LIN {X 0,Y 84.435,Z 449.066,A -85,B 0,C 180,E1 -28060.558,E2 -28060.558} C_VEL
LIN {X 0,Y 93.266,Z 446.921,A -85,B 0,C 180,E1 -28068.394,E2 -28068.394} C_VEL
LIN {X 0,Y 102.413,Z 443.94,A -85,B 0,C 180,E1 -28074.267,E2 -28074.267} C_VEL
LIN {X 0,Y 114.487,Z 439.001,A -85,B 0,C 180,E1 -28080.004,E2 -28080.004} C_VEL
LIN {X 0,Y 126.871,Z 432.782,A -85,B 0,C 180,E1 -28084.39,E2 -28084.39} C_VEL
LIN {X 0,Y 138.251,Z 425.939,A -85,B 0,C 180,E1 -28087.588,E2 -28087.588} C_VEL
LIN {X 0,Y 142.198,Z 423.34,A -85,B 0,C 180,E1 -28088.53,E2 -28088.53} C_VEL
LIN {X 0,Y 144.172,Z 421.915,A -85,B 0,C 180,E1 -28089.196,E2 -28089.196} C_VEL
LIN {X 0,Y 144.424,Z 421.642,A -85,B 0,C 180,E1 -28091.227,E2 -28091.227} C_VEL
LIN {X 0,Y 144.055,Z 421.993,A -85,B 0,C 180,E1 -28094.122,E2 -28094.122} C_VEL
LIN {X 0,Y 143.259,Z 423.001,A -85,B 0,C 180,E1 -28097.121,E2 -28097.121} C_VEL
LIN {X 0,Y 142.165,Z 424.543,A -85,B 0,C 180,E1 -28100.249,E2 -28100.249} C_VEL
LIN {X 0,Y 139.969,Z 426.46,A -85,B 0,C 180,E1 -28101.741,E2 -28101.741} C_VEL
LIN {X 0,Y 127.709,Z 434.572,A -85,B 0,C 180,E1 -28104.773,E2 -28104.773} C_VEL
LIN {X 0,Y 115.927,Z 441.264,A -85,B 0,C 180,E1 -28108.477,E2 -28108.477} C_VEL
LIN {X 0,Y 104.888,Z 446.652,A -85,B 0,C 180,E1 -28113.122,E2 -28113.122} C_VEL
LIN {X 0,Y 97.213,Z 449.956,A -85,B 0,C 180,E1 -28117.326,E2 -28117.326} C_VEL
LIN {X 0,Y 87.921,Z 453.371,A -85,B 0,C 180,E1 -28123.998,E2 -28123.998} C_VEL
LIN {X 0,Y 80.134,Z 455.727,A -85,B 0,C 180,E1 -28132.131,E2 -28132.131} C_VEL
LIN {X 0,Y 74.339,Z 457.09,A -85,B 0,C 180,E1 -28141.795,E2 -28141.795} C_VEL
LIN {X 0,Y 70.967,Z 457.423,A -85,B 0,C 180,E1 -28152.721,E2 -28152.721} C_VEL
LIN {X 0,Y 70.115,Z 456.671,A -85,B 0,C 180,E1 -28164.251,E2 -28164.251} C_VEL
LIN {X 0,Y 70.375,Z 455.877,A -85,B 0,C 180,E1 -28170.004,E2 -28170.004} C_VEL
LIN {X 0,Y 70.197,Z 454.698,A -85,B 0,C 180,E1 -28175.75,E2 -28175.75} C_VEL
LIN {X 0,Y 71.141,Z 451.341,A -85,B 0,C 180,E1 -28187.244,E2 -28187.244} C_VEL
LIN {X 0,Y 74.509,Z 446.636,A -85,B 0,C 180,E1 -28198.143,E2 -28198.143} C_VEL
LIN {X 0,Y 80.106,Z 440.454,A -85,B 0,C 180,E1 -28207.893,E2 -28207.893} C_VEL
LIN {X 0,Y 87.693,Z 432.656,A -85,B 0,C 180,E1 -28216.165,E2 -28216.165} C_VEL
LIN {X 0,Y 95.422,Z 424.288,A -85,B 0,C 180,E1 -28222.354,E2 -28222.354} C_VEL
LIN {X 0,Y 104.607,Z 413.774,A -85,B 0,C 180,E1 -28227.655,E2 -28227.655} C_VEL
LIN {X 0,Y 109.555,Z 407.579,A -85,B 0,C 180,E1 -28230.005,E2 -28230.005} C_VEL
LIN {X 0,Y 111.039,Z 404.584,A -85,B 0,C 180,E1 -28231.43,E2 -28231.43} C_VEL
LIN {X 0,Y 114.396,Z 395.038,A -85,B 0,C 180,E1 -28236.106,E2 -28236.106} C_VEL
LIN {X 0,Y 115,Z 392.347,A -85,B 0,C 180,E1 -28237.541,E2 -28237.541} C_VEL
LIN {X 0,Y 115.079,Z 383.981,A -85,B 0,C 180,E1 -28243.133,E2 -28243.133} C_VEL
LIN {X 0,Y 114.938,Z 378.464,A -85,B 0,C 180,E1 -28247.035,E2 -28247.035} C_VEL
LIN {X 0,Y 114.63,Z 373.213,A -85,B 0,C 180,E1 -28251.18,E2 -28251.18} C_VEL
LIN {X 0,Y 114.056,Z 367.486,A -85,B 0,C 180,E1 -28256.464,E2 -28256.464} C_VEL
LIN {X 0,Y 113.576,Z 364.537,A -85,B 0,C 180,E1 -28259.996,E2 -28259.996} C_VEL
LIN {X 0,Y 112.79,Z 361.934,A -85,B 0,C 180,E1 -28264.434,E2 -28264.434} C_VEL
LIN {X 0,Y 111.583,Z 360.171,A -85,B 0,C 180,E1 -28270.888,E2 -28270.888} C_VEL
LIN {X 0,Y 111.233,Z 359.571,A -85,B 0,C 180,E1 -28274.635,E2 -28274.635} C_VEL
LIN {X 0,Y 110.968,Z 359.662,A -85,B 0,C 180,E1 -28278.457,E2 -28278.457} C_VEL
LIN {X 0,Y 111.036,Z 361.087,A -85,B 0,C 180,E1 -28286.295,E2 -28286.295} C_VEL
LIN {X 0,Y 111.487,Z 362.203,A -85,B 0,C 180,E1 -28290.281,E2 -28290.281} C_VEL
LIN {X 0,Y 112.237,Z 364.789,A -85,B 0,C 180,E1 -28295.505,E2 -28295.505} C_VEL
LIN {X 0,Y 113.399,Z 369.059,A -85,B 0,C 180,E1 -28301.948,E2 -28301.948} C_VEL
LIN {X 0,Y 114.267,Z 372.788,A -85,B 0,C 180,E1 -28306.337,E2 -28306.337} C_VEL
LIN {X 0,Y 115.456,Z 378.791,A -85,B 0,C 180,E1 -28312.303,E2 -28312.303} C_VEL
LIN {X 0,Y 116.307,Z 385.128,A -85,B 0,C 180,E1 -28317.768,E2 -28317.768} C_VEL
LIN {X 0,Y 116.576,Z 388.345,A -85,B 0,C 180,E1 -28320.283,E2 -28320.283} C_VEL
LIN {X 0,Y 115.982,Z 390.167,A -85,B 0,C 180,E1 -28321.236,E2 -28321.236} C_VEL
LIN {X 0,Y 114.077,Z 392.752,A -85,B 0,C 180,E1 -28321.917,E2 -28321.917} C_VEL
LIN {X 0,Y 111.26,Z 395.53,A -85,B 0,C 180,E1 -28322.257,E2 -28322.257} C_VEL
LIN {X 0,Y 105.593,Z 400.429,A -85,B 0,C 180,E1 -28322.611,E2 -28322.611} C_VEL
LIN {X 0,Y 102.68,Z 403.357,A -85,B 0,C 180,E1 -28323.39,E2 -28323.39} C_VEL
LIN {X 0,Y 93.99,Z 413.25,A -85,B 0,C 180,E1 -28328.043,E2 -28328.043} C_VEL
LIN {X 0,Y 84.929,Z 422.622,A -85,B 0,C 180,E1 -28334.395,E2 -28334.395} C_VEL
LIN {X 0,Y 76.825,Z 430.56,A -85,B 0,C 180,E1 -28342.404,E2 -28342.404} C_VEL
LIN {X 0,Y 70.311,Z 436.93,A -85,B 0,C 180,E1 -28351.925,E2 -28351.925} C_VEL
LIN {X 0,Y 65.767,Z 441.73,A -85,B 0,C 180,E1 -28362.336,E2 -28362.336} C_VEL
LIN {X 0,Y 63.881,Z 444.105,A -85,B 0,C 180,E1 -28369.267,E2 -28369.267} C_VEL
LIN {X 0,Y 62.766,Z 446.112,A -85,B 0,C 180,E1 -28376.603,E2 -28376.603} C_VEL
LIN {X 0,Y 62.801,Z 448.526,A -85,B 0,C 180,E1 -28388.442,E2 -28388.442} C_VEL
LIN {X 0,Y 64.853,Z 449.915,A -85,B 0,C 180,E1 -28399.452,E2 -28399.452} C_VEL
LIN {X 0,Y 68.561,Z 450.524,A -85,B 0,C 180,E1 -28409.175,E2 -28409.175} C_VEL
LIN {X 0,Y 75.079,Z 450.236,A -85,B 0,C 180,E1 -28419.392,E2 -28419.392} C_VEL
LIN {X 0,Y 80.094,Z 449.536,A -85,B 0,C 180,E1 -28424.83,E2 -28424.83} C_VEL
LIN {X 0,Y 87.142,Z 448.045,A -85,B 0,C 180,E1 -28430.723,E2 -28430.723} C_VEL
LIN {X 0,Y 98.471,Z 444.801,A -85,B 0,C 180,E1 -28437.627,E2 -28437.627} C_VEL
LIN {X 0,Y 108.834,Z 441.008,A -85,B 0,C 180,E1 -28442.271,E2 -28442.271} C_VEL
LIN {X 0,Y 121.685,Z 435.179,A -85,B 0,C 180,E1 -28446.637,E2 -28446.637} C_VEL
LIN {X 0,Y 133.12,Z 428.918,A -85,B 0,C 180,E1 -28449.679,E2 -28449.679} C_VEL
LIN {X 0,Y 138.452,Z 425.626,A -85,B 0,C 180,E1 -28450.902,E2 -28450.902} C_VEL
LIN {X 0,Y 138.46,Z 425.624,A -85,B 0,C 180,E1 -28451.717,E2 -28451.717} C_VEL
LIN {X 0,Y 137.869,Z 426.196,A -85,B 0,C 180,E1 -28454.769,E2 -28454.769} C_VEL
LIN {X 0,Y 136.829,Z 427.379,A -85,B 0,C 180,E1 -28457.953,E2 -28457.953} C_VEL
LIN {X 0,Y 136.23,Z 428.01,A -85,B 0,C 180,E1 -28459.101,E2 -28459.101} C_VEL
LIN {X 0,Y 134.35,Z 429.323,A -85,B 0,C 180,E1 -28459.685,E2 -28459.685} C_VEL
LIN {X 0,Y 121.815,Z 436.836,A -85,B 0,C 180,E1 -28462.622,E2 -28462.622} C_VEL
LIN {X 0,Y 109.748,Z 442.965,A -85,B 0,C 180,E1 -28466.301,E2 -28466.301} C_VEL
LIN {X 0,Y 98.408,Z 447.887,A -85,B 0,C 180,E1 -28471.024,E2 -28471.024} C_VEL
LIN {X 0,Y 87.892,Z 451.729,A -85,B 0,C 180,E1 -28476.912,E2 -28476.912} C_VEL
LIN {X 0,Y 78.624,Z 454.487,A -85,B 0,C 180,E1 -28484.354,E2 -28484.354} C_VEL
LIN {X 0,Y 71.075,Z 456.19,A -85,B 0,C 180,E1 -28493.614,E2 -28493.614} C_VEL
LIN {X 0,Y 65.75,Z 456.915,A -85,B 0,C 180,E1 -28504.692,E2 -28504.692} C_VEL
LIN {X 0,Y 63.244,Z 456.628,A -85,B 0,C 180,E1 -28517.163,E2 -28517.163} C_VEL
LIN {X 0,Y 63.269,Z 455.362,A -85,B 0,C 180,E1 -28528.967,E2 -28528.967} C_VEL
LIN {X 0,Y 63.278,Z 454.973,A -85,B 0,C 180,E1 -28531.435,E2 -28531.435} C_VEL
LIN {X 0,Y 63.36,Z 452.358,A -85,B 0,C 180,E1 -28542.822,E2 -28542.822} C_VEL
LIN {X 0,Y 65.962,Z 448.192,A -85,B 0,C 180,E1 -28555.23,E2 -28555.23} C_VEL
LIN {X 0,Y 71.113,Z 442.605,A -85,B 0,C 180,E1 -28566.373,E2 -28566.373} C_VEL
LIN {X 0,Y 78.493,Z 435.471,A -85,B 0,C 180,E1 -28575.754,E2 -28575.754} C_VEL
LIN {X 0,Y 86.318,Z 427.807,A -85,B 0,C 180,E1 -28582.551,E2 -28582.551} C_VEL
LIN {X 0,Y 95.096,Z 418.555,A -85,B 0,C 180,E1 -28588.206,E2 -28588.206} C_VEL
LIN {X 0,Y 103.318,Z 409.184,A -85,B 0,C 180,E1 -28592.171,E2 -28592.171} C_VEL
LIN {X 0,Y 104.666,Z 407.393,A -85,B 0,C 180,E1 -28592.84,E2 -28592.84} C_VEL
LIN {X 0,Y 108.113,Z 399.375,A -85,B 0,C 180,E1 -28597.039,E2 -28597.039} C_VEL
LIN {X 0,Y 109.02,Z 397.059,A -85,B 0,C 180,E1 -28598.239,E2 -28598.239} C_VEL
LIN {X 0,Y 109.45,Z 395.202,A -85,B 0,C 180,E1 -28599.315,E2 -28599.315} C_VEL
LIN {X 0,Y 109.816,Z 389.011,A -85,B 0,C 180,E1 -28603.743,E2 -28603.743} C_VEL
LIN {X 0,Y 110.07,Z 382.163,A -85,B 0,C 180,E1 -28608.953,E2 -28608.953} C_VEL
LIN {X 0,Y 110.062,Z 377.813,A -85,B 0,C 180,E1 -28612.659,E2 -28612.659} C_VEL
LIN {X 0,Y 109.848,Z 372.283,A -85,B 0,C 180,E1 -28618.163,E2 -28618.163} C_VEL
LIN {X 0,Y 109.497,Z 369.596,A -85,B 0,C 180,E1 -28621.835,E2 -28621.835} C_VEL
LIN {X 0,Y 109.263,Z 368.507,A -85,B 0,C 180,E1 -28623.684,E2 -28623.684} C_VEL
LIN {X 0,Y 108.568,Z 367.207,A -85,B 0,C 180,E1 -28627.435,E2 -28627.435} C_VEL
LIN {X 0,Y 107.907,Z 366.105,A -85,B 0,C 180,E1 -28632.314,E2 -28632.314} C_VEL
LIN {X 0,Y 107.692,Z 365.766,A -85,B 0,C 180,E1 -28635.127,E2 -28635.127} C_VEL
LIN {X 0,Y 107.409,Z 365.93,A -85,B 0,C 180,E1 -28639.092,E2 -28639.092} C_VEL
LIN {X 0,Y 107.5,Z 367.459,A -85,B 0,C 180,E1 -28647.23,E2 -28647.23} C_VEL
LIN {X 0,Y 107.884,Z 369.197,A -85,B 0,C 180,E1 -28652.122,E2 -28652.122} C_VEL
LIN {X 0,Y 108.479,Z 371.709,A -85,B 0,C 180,E1 -28656.933,E2 -28656.933} C_VEL
LIN {X 0,Y 109.142,Z 375.046,A -85,B 0,C 180,E1 -28661.98,E2 -28661.98} C_VEL
LIN {X 0,Y 109.866,Z 379.541,A -85,B 0,C 180,E1 -28667.352,E2 -28667.352} C_VEL
LIN {X 0,Y 110.51,Z 384.899,A -85,B 0,C 180,E1 -28672.788,E2 -28672.788} C_VEL
LIN {X 0,Y 110.898,Z 390.369,A -85,B 0,C 180,E1 -28677.745,E2 -28677.745} C_VEL
LIN {X 0,Y 110.948,Z 392.488,A -85,B 0,C 180,E1 -28679.549,E2 -28679.549} C_VEL
LIN {X 0,Y 106.792,Z 398.244,A -85,B 0,C 180,E1 -28681.499,E2 -28681.499} C_VEL
LIN {X 0,Y 102.68,Z 403.357,A -85,B 0,C 180,E1 -28683.39,E2 -28683.39} C_VEL
LIN {X 0,Y 98.976,Z 407.288,A -85,B 0,C 180,E1 -28684.753,E2 -28684.753} C_VEL
LIN {X 0,Y 91.631,Z 413.346,A -85,B 0,C 180,E1 -28686.431,E2 -28686.431} C_VEL
LIN {X 0,Y 84.102,Z 418.989,A -85,B 0,C 180,E1 -28688.532,E2 -28688.532} C_VEL
LIN {X 0,Y 80.223,Z 422.232,A -85,B 0,C 180,E1 -28690.666,E2 -28690.666} C_VEL
LIN {X 0,Y 71.548,Z 430.198,A -85,B 0,C 180,E1 -28698.666,E2 -28698.666} C_VEL
LIN {X 0,Y 65.295,Z 435.825,A -85,B 0,C 180,E1 -28706.911,E2 -28706.911} C_VEL
LIN {X 0,Y 60.404,Z 440.436,A -85,B 0,C 180,E1 -28716.677,E2 -28716.677} C_VEL
LIN {X 0,Y 56.94,Z 444.245,A -85,B 0,C 180,E1 -28727.968,E2 -28727.968} C_VEL
LIN {X 0,Y 55.419,Z 447.223,A -85,B 0,C 180,E1 -28740.476,E2 -28740.476} C_VEL
LIN {X 0,Y 55.969,Z 449.038,A -85,B 0,C 180,E1 -28751.126,E2 -28751.126} C_VEL
LIN {X 0,Y 59.505,Z 450.641,A -85,B 0,C 180,E1 -28765.758,E2 -28765.758} C_VEL
LIN {X 0,Y 63.082,Z 451.003,A -85,B 0,C 180,E1 -28773.544,E2 -28773.544} C_VEL
LIN {X 0,Y 68.931,Z 450.835,A -85,B 0,C 180,E1 -28782.196,E2 -28782.196} C_VEL
LIN {X 0,Y 78.225,Z 449.653,A -85,B 0,C 180,E1 -28791.195,E2 -28791.195} C_VEL
LIN {X 0,Y 84.571,Z 448.377,A -85,B 0,C 180,E1 -28795.683,E2 -28795.683} C_VEL
LIN {X 0,Y 92.271,Z 446.416,A -85,B 0,C 180,E1 -28800.005,E2 -28800.005} C_VEL
LIN {X 0,Y 101.268,Z 443.618,A -85,B 0,C 180,E1 -28803.984,E2 -28803.984} C_VEL
LIN {X 0,Y 113.609,Z 438.825,A -85,B 0,C 180,E1 -28808.217,E2 -28808.217} C_VEL
LIN {X 0,Y 127.424,Z 432.18,A -85,B 0,C 180,E1 -28811.777,E2 -28811.777} C_VEL
LIN {X 0,Y 130.443,Z 430.488,A -85,B 0,C 180,E1 -28812.449,E2 -28812.449} C_VEL
LIN {X 0,Y 132.034,Z 429.617,A -85,B 0,C 180,E1 -28813.258,E2 -28813.258} C_VEL
LIN {X 0,Y 131.347,Z 430.27,A -85,B 0,C 180,E1 -28815.616,E2 -28815.616} C_VEL
LIN {X 0,Y 130.943,Z 430.7,A -85,B 0,C 180,E1 -28816.9,E2 -28816.9} C_VEL
LIN {X 0,Y 122.449,Z 435.584,A -85,B 0,C 180,E1 -28818.741,E2 -28818.741} C_VEL
LIN {X 0,Y 109.858,Z 441.845,A -85,B 0,C 180,E1 -28821.941,E2 -28821.941} C_VEL
LIN {X 0,Y 97.812,Z 446.907,A -85,B 0,C 180,E1 -28826.091,E2 -28826.091} C_VEL
LIN {X 0,Y 83.782,Z 451.635,A -85,B 0,C 180,E1 -28832.988,E2 -28832.988} C_VEL
LIN {X 0,Y 73.799,Z 454.277,A -85,B 0,C 180,E1 -28840.378,E2 -28840.378} C_VEL
LIN {X 0,Y 65.432,Z 455.854,A -85,B 0,C 180,E1 -28849.881,E2 -28849.881} C_VEL
LIN {X 0,Y 59.347,Z 456.429,A -85,B 0,C 180,E1 -28861.732,E2 -28861.732} C_VEL
LIN {X 0,Y 56.308,Z 456.029,A -85,B 0,C 180,E1 -28875.55,E2 -28875.55} C_VEL
LIN {X 0,Y 55.963,Z 455.433,A -85,B 0,C 180,E1 -28882.791,E2 -28882.791} C_VEL
LIN {X 0,Y 56.231,Z 454.518,A -85,B 0,C 180,E1 -28890.005,E2 -28890.005} C_VEL
LIN {X 0,Y 56.012,Z 453.189,A -85,B 0,C 180,E1 -28897.213,E2 -28897.213} C_VEL
LIN {X 0,Y 57.652,Z 449.55,A -85,B 0,C 180,E1 -28911.456,E2 -28911.456} C_VEL
LIN {X 0,Y 62.206,Z 444.536,A -85,B 0,C 180,E1 -28924.4,E2 -28924.4} C_VEL
LIN {X 0,Y 69.338,Z 438.038,A -85,B 0,C 180,E1 -28935.2,E2 -28935.2} C_VEL
LIN {X 0,Y 78.408,Z 429.881,A -85,B 0,C 180,E1 -28943.781,E2 -28943.781} C_VEL
LIN {X 0,Y 87.349,Z 421.109,A -85,B 0,C 180,E1 -28949.881,E2 -28949.881} C_VEL
LIN {X 0,Y 97.253,Z 410.652,A -85,B 0,C 180,E1 -28954.598,E2 -28954.598} C_VEL
LIN {X 0,Y 98.701,Z 409.013,A -85,B 0,C 180,E1 -28955.215,E2 -28955.215} C_VEL
LIN {X 0,Y 99.978,Z 407.155,A -85,B 0,C 180,E1 -28956.048,E2 -28956.048} C_VEL
LIN {X 0,Y 103.355,Z 399.779,A -85,B 0,C 180,E1 -28960.119,E2 -28960.119} C_VEL
LIN {X 0,Y 103.926,Z 397.995,A -85,B 0,C 180,E1 -28961.226,E2 -28961.226} C_VEL
LIN {X 0,Y 104.85,Z 390.093,A -85,B 0,C 180,E1 -28967.414,E2 -28967.414} C_VEL
LIN {X 0,Y 105.332,Z 384.283,A -85,B 0,C 180,E1 -28972.327,E2 -28972.327} C_VEL
LIN {X 0,Y 105.52,Z 379.048,A -85,B 0,C 180,E1 -28977.56,E2 -28977.56} C_VEL
LIN {X 0,Y 105.567,Z 376.988,A -85,B 0,C 180,E1 -28979.996,E2 -28979.996} C_VEL
LIN {X 0,Y 105.304,Z 374.531,A -85,B 0,C 180,E1 -28983.823,E2 -28983.823} C_VEL
LIN {X 0,Y 104.738,Z 373.153,A -85,B 0,C 180,E1 -28987.708,E2 -28987.708} C_VEL
LIN {X 0,Y 104.24,Z 372.25,A -85,B 0,C 180,E1 -28991.665,E2 -28991.665} C_VEL
LIN {X 0,Y 103.9,Z 371.842,A -85,B 0,C 180,E1 -28995.694,E2 -28995.694} C_VEL
LIN {X 0,Y 103.586,Z 372.099,A -85,B 0,C 180,E1 -28999.826,E2 -28999.826} C_VEL
LIN {X 0,Y 103.496,Z 372.773,A -85,B 0,C 180,E1 -29004.039,E2 -29004.039} C_VEL
LIN {X 0,Y 103.646,Z 373.83,A -85,B 0,C 180,E1 -29008.332,E2 -29008.332} C_VEL
LIN {X 0,Y 103.869,Z 375.502,A -85,B 0,C 180,E1 -29012.767,E2 -29012.767} C_VEL
LIN {X 0,Y 104.28,Z 377.851,A -85,B 0,C 180,E1 -29017.335,E2 -29017.335} C_VEL
LIN {X 0,Y 104.682,Z 381.147,A -85,B 0,C 180,E1 -29022.392,E2 -29022.392} C_VEL
LIN {X 0,Y 105.064,Z 385.768,A -85,B 0,C 180,E1 -29028.012,E2 -29028.012} C_VEL
LIN {X 0,Y 105.283,Z 390.711,A -85,B 0,C 180,E1 -29033.222,E2 -29033.222} C_VEL
LIN {X 0,Y 105.351,Z 394.223,A -85,B 0,C 180,E1 -29036.608,E2 -29036.608} C_VEL
LIN {X 0,Y 104.687,Z 395.748,A -85,B 0,C 180,E1 -29037.513,E2 -29037.513} C_VEL
LIN {X 0,Y 96.295,Z 405.851,A -85,B 0,C 180,E1 -29041.13,E2 -29041.13} C_VEL
LIN {X 0,Y 86.867,Z 415.825,A -85,B 0,C 180,E1 -29046.135,E2 -29046.135} C_VEL
LIN {X 0,Y 80.223,Z 422.232,A -85,B 0,C 180,E1 -29050.666,E2 -29050.666} C_VEL
LIN {X 0,Y 76.397,Z 425.363,A -85,B 0,C 180,E1 -29053.053,E2 -29053.053} C_VEL
LIN {X 0,Y 68.927,Z 430.086,A -85,B 0,C 180,E1 -29056.611,E2 -29056.611} C_VEL
LIN {X 0,Y 61.605,Z 434.373,A -85,B 0,C 180,E1 -29061.166,E2 -29061.166} C_VEL
LIN {X 0,Y 58.221,Z 436.77,A -85,B 0,C 180,E1 -29065.209,E2 -29065.209} C_VEL
LIN {X 0,Y 52.384,Z 441.9,A -85,B 0,C 180,E1 -29077.705,E2 -29077.705} C_VEL
LIN {X 0,Y 49.132,Z 445.472,A -85,B 0,C 180,E1 -29090.947,E2 -29090.947} C_VEL
LIN {X 0,Y 48.383,Z 448.247,A -85,B 0,C 180,E1 -29105.516,E2 -29105.516} C_VEL
LIN {X 0,Y 49.391,Z 449.626,A -85,B 0,C 180,E1 -29115.346,E2 -29115.346} C_VEL
LIN {X 0,Y 52.67,Z 450.886,A -85,B 0,C 180,E1 -29127.752,E2 -29127.752} C_VEL
LIN {X 0,Y 59.472,Z 451.487,A -85,B 0,C 180,E1 -29140.962,E2 -29140.962} C_VEL
LIN {X 0,Y 64.777,Z 451.319,A -85,B 0,C 180,E1 -29147.523,E2 -29147.523} C_VEL
LIN {X 0,Y 72.55,Z 450.542,A -85,B 0,C 180,E1 -29154.447,E2 -29154.447} C_VEL
LIN {X 0,Y 84.371,Z 448.357,A -85,B 0,C 180,E1 -29161.777,E2 -29161.777} C_VEL
LIN {X 0,Y 95.515,Z 445.416,A -85,B 0,C 180,E1 -29166.65,E2 -29166.65} C_VEL
LIN {X 0,Y 109.456,Z 440.593,A -85,B 0,C 180,E1 -29171.11,E2 -29171.11} C_VEL
LIN {X 0,Y 123.343,Z 434.472,A -85,B 0,C 180,E1 -29174.395,E2 -29174.395} C_VEL
LIN {X 0,Y 123.652,Z 434.376,A -85,B 0,C 180,E1 -29174.942,E2 -29174.942} C_VEL
LIN {X 0,Y 110.612,Z 440.767,A -85,B 0,C 180,E1 -29177.633,E2 -29177.633} C_VEL
LIN {X 0,Y 97.95,Z 445.937,A -85,B 0,C 180,E1 -29181.139,E2 -29181.139} C_VEL
LIN {X 0,Y 85.899,Z 449.964,A -85,B 0,C 180,E1 -29185.851,E2 -29185.851} C_VEL
LIN {X 0,Y 74.594,Z 452.919,A -85,B 0,C 180,E1 -29192.017,E2 -29192.017} C_VEL
LIN {X 0,Y 62.637,Z 455.15,A -85,B 0,C 180,E1 -29202.324,E2 -29202.324} C_VEL
LIN {X 0,Y 56.324,Z 455.855,A -85,B 0,C 180,E1 -29211.406,E2 -29211.406} C_VEL
LIN {X 0,Y 50.841,Z 455.793,A -85,B 0,C 180,E1 -29225.506,E2 -29225.506} C_VEL
LIN {X 0,Y 48.9,Z 454.745,A -85,B 0,C 180,E1 -29241.742,E2 -29241.742} C_VEL
LIN {X 0,Y 49.138,Z 453.807,A -85,B 0,C 180,E1 -29250.006,E2 -29250.006} C_VEL
LIN {X 0,Y 49.548,Z 450.682,A -85,B 0,C 180,E1 -29266.486,E2 -29266.486} C_VEL
LIN {X 0,Y 53.352,Z 446.208,A -85,B 0,C 180,E1 -29281.803,E2 -29281.803} C_VEL
LIN {X 0,Y 60.177,Z 440.3,A -85,B 0,C 180,E1 -29294.493,E2 -29294.493} C_VEL
LIN {X 0,Y 69.234,Z 432.816,A -85,B 0,C 180,E1 -29304.307,E2 -29304.307} C_VEL
LIN {X 0,Y 78.401,Z 424.767,A -85,B 0,C 180,E1 -29310.935,E2 -29310.935} C_VEL
LIN {X 0,Y 86.771,Z 416.714,A -85,B 0,C 180,E1 -29315.425,E2 -29315.425} C_VEL
LIN {X 0,Y 94.36,Z 408.728,A -85,B 0,C 180,E1 -29318.6,E2 -29318.6} C_VEL
LIN {X 0,Y 98.056,Z 401.838,A -85,B 0,C 180,E1 -29322.567,E2 -29322.567} C_VEL
LIN {X 0,Y 98.683,Z 399.29,A -85,B 0,C 180,E1 -29324.506,E2 -29324.506} C_VEL
LIN {X 0,Y 99.861,Z 392.639,A -85,B 0,C 180,E1 -29330.174,E2 -29330.174} C_VEL
LIN {X 0,Y 100.481,Z 388.551,A -85,B 0,C 180,E1 -29333.973,E2 -29333.973} C_VEL
LIN {X 0,Y 101.088,Z 383.061,A -85,B 0,C 180,E1 -29339.996,E2 -29339.996} C_VEL
LIN {X 0,Y 101.104,Z 380.39,A -85,B 0,C 180,E1 -29343.982,E2 -29343.982} C_VEL
LIN {X 0,Y 100.672,Z 378.954,A -85,B 0,C 180,E1 -29348.022,E2 -29348.022} C_VEL
LIN {X 0,Y 100.212,Z 378.082,A -85,B 0,C 180,E1 -29352.141,E2 -29352.141} C_VEL
LIN {X 0,Y 99.881,Z 377.758,A -85,B 0,C 180,E1 -29356.342,E2 -29356.342} C_VEL
LIN {X 0,Y 99.438,Z 378.508,A -85,B 0,C 180,E1 -29363.242,E2 -29363.242} C_VEL
LIN {X 0,Y 99.491,Z 380.153,A -85,B 0,C 180,E1 -29369.63,E2 -29369.63} C_VEL
LIN {X 0,Y 99.638,Z 382.034,A -85,B 0,C 180,E1 -29374.347,E2 -29374.347} C_VEL
LIN {X 0,Y 99.868,Z 384.755,A -85,B 0,C 180,E1 -29379.292,E2 -29379.292} C_VEL
LIN {X 0,Y 99.952,Z 389.013,A -85,B 0,C 180,E1 -29385.317,E2 -29385.317} C_VEL
LIN {X 0,Y 99.916,Z 393.541,A -85,B 0,C 180,E1 -29390.721,E2 -29390.721} C_VEL
LIN {X 0,Y 99.77,Z 397.024,A -85,B 0,C 180,E1 -29394.469,E2 -29394.469} C_VEL
LIN {X 0,Y 92.047,Z 406.035,A -85,B 0,C 180,E1 -29397.689,E2 -29397.689} C_VEL
LIN {X 0,Y 82.829,Z 415.378,A -85,B 0,C 180,E1 -29402.178,E2 -29402.178} C_VEL
LIN {X 0,Y 72.804,Z 424.53,A -85,B 0,C 180,E1 -29408.773,E2 -29408.773} C_VEL
LIN {X 0,Y 63.883,Z 432.065,A -85,B 0,C 180,E1 -29417.285,E2 -29417.285} C_VEL
LIN {X 0,Y 58.221,Z 436.77,A -85,B 0,C 180,E1 -29425.209,E2 -29425.209} C_VEL
LIN {X 0,Y 55.065,Z 439.039,A -85,B 0,C 180,E1 -29429.726,E2 -29429.726} C_VEL
LIN {X 0,Y 48.756,Z 442.277,A -85,B 0,C 180,E1 -29437.399,E2 -29437.399} C_VEL
LIN {X 0,Y 44.11,Z 444.57,A -85,B 0,C 180,E1 -29444.982,E2 -29444.982} C_VEL
LIN {X 0,Y 41.881,Z 446.093,A -85,B 0,C 180,E1 -29452.067,E2 -29452.067} C_VEL
LIN {X 0,Y 41.535,Z 446.597,A -85,B 0,C 180,E1 -29454.663,E2 -29454.663} C_VEL
LIN {X 0,Y 42.751,Z 450.019,A -85,B 0,C 180,E1 -29478.898,E2 -29478.898} C_VEL
LIN {X 0,Y 47.137,Z 451.365,A -85,B 0,C 180,E1 -29493.441,E2 -29493.441} C_VEL
LIN {X 0,Y 53.449,Z 451.966,A -85,B 0,C 180,E1 -29504.762,E2 -29504.762} C_VEL
LIN {X 0,Y 63.45,Z 451.685,A -85,B 0,C 180,E1 -29515.419,E2 -29515.419} C_VEL
LIN {X 0,Y 70.276,Z 450.99,A -85,B 0,C 180,E1 -29520.367,E2 -29520.367} C_VEL
LIN {X 0,Y 78.928,Z 449.597,A -85,B 0,C 180,E1 -29525.114,E2 -29525.114} C_VEL
LIN {X 0,Y 92.962,Z 446.337,A -85,B 0,C 180,E1 -29530.656,E2 -29530.656} C_VEL
LIN {X 0,Y 105.754,Z 442.311,A -85,B 0,C 180,E1 -29534.265,E2 -29534.265} C_VEL
LIN {X 0,Y 103.4,Z 443.247,A -85,B 0,C 180,E1 -29535.185,E2 -29535.185} C_VEL
LIN {X 0,Y 89.254,Z 448.158,A -85,B 0,C 180,E1 -29539.119,E2 -29539.119} C_VEL
LIN {X 0,Y 76.922,Z 451.501,A -85,B 0,C 180,E1 -29543.994,E2 -29543.994} C_VEL
LIN {X 0,Y 65.427,Z 453.788,A -85,B 0,C 180,E1 -29550.766,E2 -29550.766} C_VEL
LIN {X 0,Y 55.238,Z 455.114,A -85,B 0,C 180,E1 -29560.245,E2 -29560.245} C_VEL
LIN {X 0,Y 47.22,Z 455.455,A -85,B 0,C 180,E1 -29573.47,E2 -29573.47} C_VEL
LIN {X 0,Y 42.618,Z 454.757,A -85,B 0,C 180,E1 -29590.749,E2 -29590.749} C_VEL
LIN {X 0,Y 41.879,Z 454.035,A -85,B 0,C 180,E1 -29600.346,E2 -29600.346} C_VEL
LIN {X 0,Y 42.047,Z 453.032,A -85,B 0,C 180,E1 -29610.007,E2 -29610.007} C_VEL
LIN {X 0,Y 42.751,Z 449.8,A -85,B 0,C 180,E1 -29629.202,E2 -29629.202} C_VEL
LIN {X 0,Y 47.405,Z 445.193,A -85,B 0,C 180,E1 -29646.378,E2 -29646.378} C_VEL
LIN {X 0,Y 55.291,Z 439.121,A -85,B 0,C 180,E1 -29659.706,E2 -29659.706} C_VEL
LIN {X 0,Y 65.321,Z 431.452,A -85,B 0,C 180,E1 -29669.408,E2 -29669.408} C_VEL
LIN {X 0,Y 75.151,Z 423.192,A -85,B 0,C 180,E1 -29675.765,E2 -29675.765} C_VEL
LIN {X 0,Y 85.054,Z 413.964,A -85,B 0,C 180,E1 -29680.255,E2 -29680.255} C_VEL
LIN {X 0,Y 89.872,Z 408.991,A -85,B 0,C 180,E1 -29682.063,E2 -29682.063} C_VEL
LIN {X 0,Y 92.314,Z 404.87,A -85,B 0,C 180,E1 -29684.582,E2 -29684.582} C_VEL
LIN {X 0,Y 93.072,Z 403.185,A -85,B 0,C 180,E1 -29685.809,E2 -29685.809} C_VEL
LIN {X 0,Y 94.58,Z 397.023,A -85,B 0,C 180,E1 -29691.449,E2 -29691.449} C_VEL
LIN {X 0,Y 95.568,Z 392.667,A -85,B 0,C 180,E1 -29695.778,E2 -29695.778} C_VEL
LIN {X 0,Y 96.305,Z 388.994,A -85,B 0,C 180,E1 -29699.996,E2 -29699.996} C_VEL
LIN {X 0,Y 96.65,Z 386.102,A -85,B 0,C 180,E1 -29704.166,E2 -29704.166} C_VEL
LIN {X 0,Y 96.372,Z 384.584,A -85,B 0,C 180,E1 -29708.382,E2 -29708.382} C_VEL
LIN {X 0,Y 95.948,Z 383.771,A -85,B 0,C 180,E1 -29712.689,E2 -29712.689} C_VEL
LIN {X 0,Y 95.593,Z 383.573,A -85,B 0,C 180,E1 -29717.097,E2 -29717.097} C_VEL
LIN {X 0,Y 95.225,Z 384,A -85,B 0,C 180,E1 -29721.65,E2 -29721.65} C_VEL
LIN {X 0,Y 95.065,Z 385.249,A -85,B 0,C 180,E1 -29727.479,E2 -29727.479} C_VEL
LIN {X 0,Y 95.091,Z 386.337,A -85,B 0,C 180,E1 -29731.149,E2 -29731.149} C_VEL
LIN {X 0,Y 95.059,Z 388.584,A -85,B 0,C 180,E1 -29736.255,E2 -29736.255} C_VEL
LIN {X 0,Y 94.943,Z 391.861,A -85,B 0,C 180,E1 -29741.769,E2 -29741.769} C_VEL
LIN {X 0,Y 94.645,Z 396.492,A -85,B 0,C 180,E1 -29748.059,E2 -29748.059} C_VEL
LIN {X 0,Y 94.411,Z 398.442,A -85,B 0,C 180,E1 -29750.429,E2 -29750.429} C_VEL
LIN {X 0,Y 93.991,Z 399.827,A -85,B 0,C 180,E1 -29751.753,E2 -29751.753} C_VEL
LIN {X 0,Y 84.005,Z 410.368,A -85,B 0,C 180,E1 -29755.613,E2 -29755.613} C_VEL
LIN {X 0,Y 74.529,Z 419.129,A -85,B 0,C 180,E1 -29760.322,E2 -29760.322} C_VEL
LIN {X 0,Y 64.272,Z 427.668,A -85,B 0,C 180,E1 -29767.493,E2 -29767.493} C_VEL
LIN {X 0,Y 56.311,Z 433.814,A -85,B 0,C 180,E1 -29775.54,E2 -29775.54} C_VEL
LIN {X 0,Y 49.279,Z 439.196,A -85,B 0,C 180,E1 -29786.51,E2 -29786.51} C_VEL
LIN {X 0,Y 43.331,Z 444.274,A -85,B 0,C 180,E1 -29803.35,E2 -29803.35} C_VEL
LIN {X 0,Y 41.535,Z 446.597,A -85,B 0,C 180,E1 -29814.663,E2 -29814.663} C_VEL
LIN {X 0,Y 40.534,Z 447.996,A -85,B 0,C 180,E1 -29822.558,E2 -29822.558} C_VEL
LIN {X 0,Y 38.666,Z 449.813,A -85,B 0,C 180,E1 -29836.45,E2 -29836.45} C_VEL
LIN {X 0,Y 38.654,Z 450.887,A -85,B 0,C 180,E1 -29848.231,E2 -29848.231} C_VEL
LIN {X 0,Y 40.38,Z 451.536,A -85,B 0,C 180,E1 -29856.462,E2 -29856.462} C_VEL
LIN {X 0,Y 41.356,Z 451.707,A -85,B 0,C 180,E1 -29858.875,E2 -29858.875} C_VEL
LIN {X 0,Y 49.682,Z 452.449,A -85,B 0,C 180,E1 -29871.938,E2 -29871.938} C_VEL
LIN {X 0,Y 58.276,Z 452.31,A -85,B 0,C 180,E1 -29880.007,E2 -29880.007} C_VEL
LIN {X 0,Y 70.904,Z 451.145,A -85,B 0,C 180,E1 -29887.638,E2 -29887.638} C_VEL
LIN {X 0,Y 78.738,Z 449.893,A -85,B 0,C 180,E1 -29890.957,E2 -29890.957} C_VEL
LIN {X 0,Y 87.584,Z 448.042,A -85,B 0,C 180,E1 -29893.934,E2 -29893.934} C_VEL
LIN {X 0,Y 87.176,Z 448.212,A -85,B 0,C 180,E1 -29894.678,E2 -29894.678} C_VEL
LIN {X 0,Y 74.299,Z 451.4,A -85,B 0,C 180,E1 -29898.945,E2 -29898.945} C_VEL
LIN {X 0,Y 62.072,Z 453.55,A -85,B 0,C 180,E1 -29905.082,E2 -29905.082} C_VEL
LIN {X 0,Y 50.888,Z 454.706,A -85,B 0,C 180,E1 -29914.05,E2 -29914.05} C_VEL
LIN {X 0,Y 41.687,Z 454.925,A -85,B 0,C 180,E1 -29927.605,E2 -29927.605} C_VEL
LIN {X 0,Y 35.966,Z 454.117,A -85,B 0,C 180,E1 -29947.003,E2 -29947.003} C_VEL
LIN {X 0,Y 34.939,Z 452.234,A -85,B 0,C 180,E1 -29970.008,E2 -29970.008} C_VEL
LIN {X 0,Y 36.097,Z 448.836,A -85,B 0,C 180,E1 -29992.925,E2 -29992.925} C_VEL
LIN {X 0,Y 41.852,Z 444.066,A -85,B 0,C 180,E1 -30012.207,E2 -30012.207} C_VEL
LIN {X 0,Y 50.946,Z 437.826,A -85,B 0,C 180,E1 -30025.872,E2 -30025.872} C_VEL
LIN {X 0,Y 61.974,Z 429.95,A -85,B 0,C 180,E1 -30035.133,E2 -30035.133} C_VEL
LIN {X 0,Y 72.477,Z 421.492,A -85,B 0,C 180,E1 -30040.998,E2 -30040.998} C_VEL
LIN {X 0,Y 82.163,Z 412.814,A -85,B 0,C 180,E1 -30044.682,E2 -30044.682} C_VEL
LIN {X 0,Y 85.355,Z 409.64,A -85,B 0,C 180,E1 -30045.694,E2 -30045.694} C_VEL
LIN {X 0,Y 87.665,Z 405.969,A -85,B 0,C 180,E1 -30048.158,E2 -30048.158} C_VEL
LIN {X 0,Y 89.701,Z 399.76,A -85,B 0,C 180,E1 -30054.375,E2 -30054.375} C_VEL
LIN {X 0,Y 91.186,Z 394.802,A -85,B 0,C 180,E1 -30059.995,E2 -30059.995} C_VEL
LIN {X 0,Y 91.909,Z 391.697,A -85,B 0,C 180,E1 -30064.381,E2 -30064.381} C_VEL
LIN {X 0,Y 91.853,Z 390.038,A -85,B 0,C 180,E1 -30068.798,E2 -30068.798} C_VEL
LIN {X 0,Y 91.458,Z 389.299,A -85,B 0,C 180,E1 -30073.323,E2 -30073.323} C_VEL
LIN {X 0,Y 91.056,Z 389.248,A -85,B 0,C 180,E1 -30077.978,E2 -30077.978} C_VEL
LIN {X 0,Y 90.642,Z 389.789,A -85,B 0,C 180,E1 -30082.805,E2 -30082.805} C_VEL
LIN {X 0,Y 90.477,Z 390.835,A -85,B 0,C 180,E1 -30087.773,E2 -30087.773} C_VEL
LIN {X 0,Y 90.263,Z 392.616,A -85,B 0,C 180,E1 -30093.021,E2 -30093.021} C_VEL
LIN {X 0,Y 90.191,Z 393.678,A -85,B 0,C 180,E1 -30095.576,E2 -30095.576} C_VEL
LIN {X 0,Y 90.013,Z 395.309,A -85,B 0,C 180,E1 -30098.664,E2 -30098.664} C_VEL
LIN {X 0,Y 89.423,Z 399.309,A -85,B 0,C 180,E1 -30105.011,E2 -30105.011} C_VEL
LIN {X 0,Y 89.132,Z 401.074,A -85,B 0,C 180,E1 -30107.404,E2 -30107.404} C_VEL
LIN {X 0,Y 88.189,Z 402.67,A -85,B 0,C 180,E1 -30108.637,E2 -30108.637} C_VEL
LIN {X 0,Y 77.771,Z 412.91,A -85,B 0,C 180,E1 -30112.407,E2 -30112.407} C_VEL
LIN {X 0,Y 67.913,Z 421.368,A -85,B 0,C 180,E1 -30117.087,E2 -30117.087} C_VEL
LIN {X 0,Y 57.154,Z 429.604,A -85,B 0,C 180,E1 -30124.503,E2 -30124.503} C_VEL
LIN {X 0,Y 48.754,Z 435.473,A -85,B 0,C 180,E1 -30133.238,E2 -30133.238} C_VEL
LIN {X 0,Y 42.433,Z 439.897,A -85,B 0,C 180,E1 -30143.493,E2 -30143.493} C_VEL
LIN {X 0,Y 36.018,Z 444.851,A -85,B 0,C 180,E1 -30162.735,E2 -30162.735} C_VEL
LIN {X 0,Y 34.231,Z 448.668,A -85,B 0,C 180,E1 -30188.01,E2 -30188.01} C_VEL
LIN {X 0,Y 36.6,Z 450.497,A -85,B 0,C 180,E1 -30204.84,E2 -30204.84} C_VEL
LIN {X 0,Y 41.356,Z 451.707,A -85,B 0,C 180,E1 -30218.875,E2 -30218.875} C_VEL
LIN {X 0,Y 44.267,Z 452.204,A -85,B 0,C 180,E1 -30225.724,E2 -30225.724} C_VEL
LIN {X 0,Y 48.822,Z 452.744,A -85,B 0,C 180,E1 -30236.573,E2 -30236.573} C_VEL
LIN {X 0,Y 53.382,Z 452.872,A -85,B 0,C 180,E1 -30243.907,E2 -30243.907} C_VEL
LIN {X 0,Y 57.78,Z 452.738,A -85,B 0,C 180,E1 -30248.005,E2 -30248.005} C_VEL
LIN {X 0,Y 59.453,Z 452.596,A -85,B 0,C 180,E1 -30249.026,E2 -30249.026} C_VEL
LIN {X 0,Y 69.222,Z 451.756,A -85,B 0,C 180,E1 -30253.413,E2 -30253.413} C_VEL
LIN {X 0,Y 65.773,Z 452.403,A -85,B 0,C 180,E1 -30255.93,E2 -30255.93} C_VEL
LIN {X 0,Y 53.19,Z 453.93,A -85,B 0,C 180,E1 -30262.359,E2 -30262.359} C_VEL
LIN {X 0,Y 41.709,Z 454.443,A -85,B 0,C 180,E1 -30272.607,E2 -30272.607} C_VEL
LIN {X 0,Y 32.571,Z 454.027,A -85,B 0,C 180,E1 -30289.671,E2 -30289.671} C_VEL
LIN {X 0,Y 27.953,Z 452.594,A -85,B 0,C 180,E1 -30315.448,E2 -30315.448} C_VEL
LIN {X 0,Y 27.844,Z 451.44,A -85,B 0,C 180,E1 -30330.01,E2 -30330.01} C_VEL
LIN {X 0,Y 29.667,Z 447.874,A -85,B 0,C 180,E1 -30358.291,E2 -30358.291} C_VEL
LIN {X 0,Y 36.862,Z 442.922,A -85,B 0,C 180,E1 -30379.708,E2 -30379.708} C_VEL
LIN {X 0,Y 47.283,Z 436.488,A -85,B 0,C 180,E1 -30393.116,E2 -30393.116} C_VEL
LIN {X 0,Y 59.313,Z 428.411,A -85,B 0,C 180,E1 -30401.442,E2 -30401.442} C_VEL
LIN {X 0,Y 70.462,Z 419.719,A -85,B 0,C 180,E1 -30406.543,E2 -30406.543} C_VEL
LIN {X 0,Y 80.818,Z 410.574,A -85,B 0,C 180,E1 -30409.664,E2 -30409.664} C_VEL
LIN {X 0,Y 81.603,Z 409.686,A -85,B 0,C 180,E1 -30410.076,E2 -30410.076} C_VEL
LIN {X 0,Y 82.594,Z 408.061,A -85,B 0,C 180,E1 -30411.431,E2 -30411.431} C_VEL
LIN {X 0,Y 84.866,Z 402.619,A -85,B 0,C 180,E1 -30417.384,E2 -30417.384} C_VEL
LIN {X 0,Y 86.379,Z 398.67,A -85,B 0,C 180,E1 -30422.327,E2 -30422.327} C_VEL
LIN {X 0,Y 86.891,Z 396.876,A -85,B 0,C 180,E1 -30425.321,E2 -30425.321} C_VEL
LIN {X 0,Y 87.139,Z 395.299,A -85,B 0,C 180,E1 -30429.278,E2 -30429.278} C_VEL
LIN {X 0,Y 86.729,Z 394.681,A -85,B 0,C 180,E1 -30434.064,E2 -30434.064} C_VEL
LIN {X 0,Y 86.292,Z 394.732,A -85,B 0,C 180,E1 -30439.007,E2 -30439.007} C_VEL
LIN {X 0,Y 85.739,Z 395.703,A -85,B 0,C 180,E1 -30445.615,E2 -30445.615} C_VEL
LIN {X 0,Y 85.573,Z 396.677,A -85,B 0,C 180,E1 -30449.517,E2 -30449.517} C_VEL
LIN {X 0,Y 85.116,Z 398.834,A -85,B 0,C 180,E1 -30455.302,E2 -30455.302} C_VEL
LIN {X 0,Y 84.335,Z 402.366,A -85,B 0,C 180,E1 -30461.803,E2 -30461.803} C_VEL
LIN {X 0,Y 83.91,Z 403.904,A -85,B 0,C 180,E1 -30464.304,E2 -30464.304} C_VEL
LIN {X 0,Y 82.464,Z 405.571,A -85,B 0,C 180,E1 -30465.169,E2 -30465.169} C_VEL
LIN {X 0,Y 71.789,Z 415.323,A -85,B 0,C 180,E1 -30468.633,E2 -30468.633} C_VEL
LIN {X 0,Y 59.903,Z 424.695,A -85,B 0,C 180,E1 -30474.078,E2 -30474.078} C_VEL
LIN {X 0,Y 48.664,Z 432.43,A -85,B 0,C 180,E1 -30482.001,E2 -30482.001} C_VEL
LIN {X 0,Y 38.563,Z 438.765,A -85,B 0,C 180,E1 -30494.128,E2 -30494.128} C_VEL
LIN {X 0,Y 31.489,Z 443.27,A -85,B 0,C 180,E1 -30509.991,E2 -30509.991} C_VEL
LIN {X 0,Y 27.378,Z 446.86,A -85,B 0,C 180,E1 -30532.636,E2 -30532.636} C_VEL
LIN {X 0,Y 28.03,Z 449.663,A -85,B 0,C 180,E1 -30558.764,E2 -30558.764} C_VEL
LIN {X 0,Y 31.26,Z 451.052,A -85,B 0,C 180,E1 -30574.046,E2 -30574.046} C_VEL
LIN {X 0,Y 38.023,Z 452.306,A -85,B 0,C 180,E1 -30589.36,E2 -30589.36} C_VEL
LIN {X 0,Y 49.23,Z 452.943,A -85,B 0,C 180,E1 -30602.279,E2 -30602.279} C_VEL
LIN {X 0,Y 59.453,Z 452.596,A -85,B 0,C 180,E1 -30609.026,E2 -30609.026} C_VEL
LIN {X 0,Y 58.47,Z 452.778,A -85,B 0,C 180,E1 -30609.534,E2 -30609.534} C_VEL
LIN {X 0,Y 52.668,Z 453.17,A -85,B 0,C 180,E1 -30608.954,E2 -30608.954} C_VEL
LIN {X 0,Y 40.072,Z 453.097,A -85,B 0,C 180,E1 -30603.599,E2 -30603.599} C_VEL
LIN {X 0,Y 34.879,Z 452.735,A -85,B 0,C 180,E1 -30599.421,E2 -30599.421} C_VEL
LIN {X 0,Y 30.219,Z 452.131,A -85,B 0,C 180,E1 -30593.181,E2 -30593.181} C_VEL
LIN {X 0,Y 23.285,Z 450.609,A -85,B 0,C 180,E1 -30574.861,E2 -30574.861} C_VEL
LIN {X 0,Y 19.915,Z 448.034,A -85,B 0,C 180,E1 -30541.945,E2 -30541.945} C_VEL
LIN {X 0,Y 23.352,Z 444.538,A -85,B 0,C 180,E1 -30509.988,E2 -30509.988} C_VEL
LIN {X 0,Y 31.638,Z 439.899,A -85,B 0,C 180,E1 -30489.058,E2 -30489.058} C_VEL
LIN {X 0,Y 41.896,Z 434.172,A -85,B 0,C 180,E1 -30476.988,E2 -30476.988} C_VEL
LIN {X 0,Y 53.834,Z 426.697,A -85,B 0,C 180,E1 -30469.245,E2 -30469.245} C_VEL
LIN {X 0,Y 66.185,Z 417.669,A -85,B 0,C 180,E1 -30464.206,E2 -30464.206} C_VEL
LIN {X 0,Y 78.653,Z 406.889,A -85,B 0,C 180,E1 -30460.789,E2 -30460.789} C_VEL
LIN {X 0,Y 79.476,Z 404.853,A -85,B 0,C 180,E1 -30457.258,E2 -30457.258} C_VEL
LIN {X 0,Y 80.232,Z 402.574,A -85,B 0,C 180,E1 -30451.7,E2 -30451.7} C_VEL
LIN {X 0,Y 80.741,Z 400.935,A -85,B 0,C 180,E1 -30445.793,E2 -30445.793} C_VEL
LIN {X 0,Y 81.485,Z 399.93,A -85,B 0,C 180,E1 -30438.414,E2 -30438.414} C_VEL
LIN {X 0,Y 81.775,Z 399.899,A -85,B 0,C 180,E1 -30434.936,E2 -30434.936} C_VEL
LIN {X 0,Y 82.212,Z 400.39,A -85,B 0,C 180,E1 -30429.839,E2 -30429.839} C_VEL
LIN {X 0,Y 81.583,Z 402.456,A -85,B 0,C 180,E1 -30424.937,E2 -30424.937} C_VEL
LIN {X 0,Y 79.867,Z 406.037,A -85,B 0,C 180,E1 -30419.995,E2 -30419.995} C_VEL
LIN {X 0,Y 77.632,Z 410.36,A -85,B 0,C 180,E1 -30414.8,E2 -30414.8} C_VEL
LIN {X 0,Y 76.371,Z 411.801,A -85,B 0,C 180,E1 -30414.019,E2 -30414.019} C_VEL
LIN {X 0,Y 65.759,Z 420.647,A -85,B 0,C 180,E1 -30411.365,E2 -30411.365} C_VEL
LIN {X 0,Y 54.143,Z 429.094,A -85,B 0,C 180,E1 -30406.808,E2 -30406.808} C_VEL
LIN {X 0,Y 41.406,Z 436.944,A -85,B 0,C 180,E1 -30399.009,E2 -30399.009} C_VEL
LIN {X 0,Y 30.071,Z 443.177,A -85,B 0,C 180,E1 -30384.9,E2 -30384.9} C_VEL
LIN {X 0,Y 22.137,Z 447.926,A -85,B 0,C 180,E1 -30358.453,E2 -30358.453} C_VEL
LIN {X 0,Y 20.739,Z 450.619,A -85,B 0,C 180,E1 -30330.013,E2 -30330.013} C_VEL
LIN {X 0,Y 21.141,Z 451.823,A -85,B 0,C 180,E1 -30310.597,E2 -30310.597} C_VEL
LIN {X 0,Y 27.509,Z 453.37,A -85,B 0,C 180,E1 -30279.981,E2 -30279.981} C_VEL
LIN {X 0,Y 38.32,Z 453.951,A -85,B 0,C 180,E1 -30263.524,E2 -30263.524} C_VEL
LIN {X 0,Y 50.894,Z 453.564,A -85,B 0,C 180,E1 -30254.862,E2 -30254.862} C_VEL
LIN {X 0,Y 51.987,Z 453.444,A -85,B 0,C 180,E1 -30253.297,E2 -30253.297} C_VEL
LIN {X 0,Y 42.517,Z 453.312,A -85,B 0,C 180,E1 -30247.4,E2 -30247.4} C_VEL
LIN {X 0,Y 30.219,Z 452.131,A -85,B 0,C 180,E1 -30233.181,E2 -30233.181} C_VEL
LIN {X 0,Y 25.721,Z 451.448,A -85,B 0,C 180,E1 -30225.458,E2 -30225.458} C_VEL
LIN {X 0,Y 18.205,Z 449.902,A -85,B 0,C 180,E1 -30208.787,E2 -30208.787} C_VEL
LIN {X 0,Y 13.995,Z 448.259,A -85,B 0,C 180,E1 -30184.931,E2 -30184.931} C_VEL
LIN {X 0,Y 13.827,Z 446.728,A -85,B 0,C 180,E1 -30161.046,E2 -30161.046} C_VEL
LIN {X 0,Y 14.506,Z 446.155,A -85,B 0,C 180,E1 -30153.855,E2 -30153.855} C_VEL
LIN {X 0,Y 23.528,Z 441.725,A -85,B 0,C 180,E1 -30123.61,E2 -30123.61} C_VEL
LIN {X 0,Y 33.856,Z 436.69,A -85,B 0,C 180,E1 -30111.472,E2 -30111.472} C_VEL
LIN {X 0,Y 46.394,Z 429.681,A -85,B 0,C 180,E1 -30103.974,E2 -30103.974} C_VEL
LIN {X 0,Y 59.2,Z 421.186,A -85,B 0,C 180,E1 -30099.49,E2 -30099.49} C_VEL
LIN {X 0,Y 71.674,Z 411.341,A -85,B 0,C 180,E1 -30096.653,E2 -30096.653} C_VEL
LIN {X 0,Y 73.016,Z 410.175,A -85,B 0,C 180,E1 -30096.393,E2 -30096.393} C_VEL
LIN {X 0,Y 74.373,Z 408.599,A -85,B 0,C 180,E1 -30094.532,E2 -30094.532} C_VEL
LIN {X 0,Y 74.782,Z 407.699,A -85,B 0,C 180,E1 -30092.234,E2 -30092.234} C_VEL
LIN {X 0,Y 75.357,Z 406.359,A -85,B 0,C 180,E1 -30087.789,E2 -30087.789} C_VEL
LIN {X 0,Y 75.938,Z 405.344,A -85,B 0,C 180,E1 -30081.721,E2 -30081.721} C_VEL
LIN {X 0,Y 76.63,Z 404.917,A -85,B 0,C 180,E1 -30075.964,E2 -30075.964} C_VEL
LIN {X 0,Y 77.073,Z 405.304,A -85,B 0,C 180,E1 -30070.502,E2 -30070.502} C_VEL
LIN {X 0,Y 76.702,Z 406.242,A -85,B 0,C 180,E1 -30067.894,E2 -30067.894} C_VEL
LIN {X 0,Y 75.907,Z 407.669,A -85,B 0,C 180,E1 -30065.307,E2 -30065.307} C_VEL
LIN {X 0,Y 73.551,Z 411.502,A -85,B 0,C 180,E1 -30059.994,E2 -30059.994} C_VEL
LIN {X 0,Y 72.162,Z 413.022,A -85,B 0,C 180,E1 -30058.836,E2 -30058.836} C_VEL
LIN {X 0,Y 61.596,Z 421.479,A -85,B 0,C 180,E1 -30056.802,E2 -30056.802} C_VEL
LIN {X 0,Y 49.541,Z 429.704,A -85,B 0,C 180,E1 -30053.282,E2 -30053.282} C_VEL
LIN {X 0,Y 36.108,Z 437.343,A -85,B 0,C 180,E1 -30046.736,E2 -30046.736} C_VEL
LIN {X 0,Y 23.66,Z 443.397,A -85,B 0,C 180,E1 -30033.039,E2 -30033.039} C_VEL
LIN {X 0,Y 14.616,Z 447.966,A -85,B 0,C 180,E1 -29998.762,E2 -29998.762} C_VEL
LIN {X 0,Y 13.627,Z 449.729,A -85,B 0,C 180,E1 -29970.02,E2 -29970.02} C_VEL
LIN {X 0,Y 14.615,Z 450.997,A -85,B 0,C 180,E1 -29941.279,E2 -29941.279} C_VEL
LIN {X 0,Y 23.564,Z 452.701,A -85,B 0,C 180,E1 -29906.548,E2 -29906.548} C_VEL
LIN {X 0,Y 29.617,Z 453.196,A -85,B 0,C 180,E1 -29898.374,E2 -29898.374} C_VEL
LIN {X 0,Y 33.208,Z 453.223,A -85,B 0,C 180,E1 -29892.231,E2 -29892.231} C_VEL
LIN {X 0,Y 21.118,Z 451.549,A -85,B 0,C 180,E1 -29876.521,E2 -29876.521} C_VEL
LIN {X 0,Y 14.494,Z 449.643,A -85,B 0,C 180,E1 -29851.03,E2 -29851.03} C_VEL
LIN {X 0,Y 14.506,Z 446.155,A -85,B 0,C 180,E1 -29793.855,E2 -29793.855} C_VEL
LIN {X 0,Y 17.221,Z 444.411,A -85,B 0,C 180,E1 -29775.924,E2 -29775.924} C_VEL
LIN {X 0,Y 22.86,Z 441.158,A -85,B 0,C 180,E1 -29754.159,E2 -29754.159} C_VEL
LIN {X 0,Y 30.141,Z 437.383,A -85,B 0,C 180,E1 -29741.607,E2 -29741.607} C_VEL
LIN {X 0,Y 35.157,Z 434.796,A -85,B 0,C 180,E1 -29738.176,E2 -29738.176} C_VEL
LIN {X 0,Y 47.043,Z 428.149,A -85,B 0,C 180,E1 -29734.766,E2 -29734.766} C_VEL
LIN {X 0,Y 60.294,Z 419.253,A -85,B 0,C 180,E1 -29732.311,E2 -29732.311} C_VEL
LIN {X 0,Y 67.515,Z 413.655,A -85,B 0,C 180,E1 -29731.356,E2 -29731.356} C_VEL
LIN {X 0,Y 69.456,Z 411.882,A -85,B 0,C 180,E1 -29730.386,E2 -29730.386} C_VEL
LIN {X 0,Y 70.137,Z 410.746,A -85,B 0,C 180,E1 -29725.591,E2 -29725.591} C_VEL
LIN {X 0,Y 71.161,Z 409.842,A -85,B 0,C 180,E1 -29717.228,E2 -29717.228} C_VEL
LIN {X 0,Y 71.713,Z 410.023,A -85,B 0,C 180,E1 -29711.297,E2 -29711.297} C_VEL
LIN {X 0,Y 70.872,Z 411.368,A -85,B 0,C 180,E1 -29708.074,E2 -29708.074} C_VEL
LIN {X 0,Y 69.861,Z 412.749,A -85,B 0,C 180,E1 -29705.767,E2 -29705.767} C_VEL
LIN {X 0,Y 68.225,Z 414.481,A -85,B 0,C 180,E1 -29704.203,E2 -29704.203} C_VEL
LIN {X 0,Y 56.295,Z 423.454,A -85,B 0,C 180,E1 -29702.774,E2 -29702.774} C_VEL
LIN {X 0,Y 43.932,Z 431.238,A -85,B 0,C 180,E1 -29700.538,E2 -29700.538} C_VEL
LIN {X 0,Y 31.679,Z 437.656,A -85,B 0,C 180,E1 -29696.84,E2 -29696.84} C_VEL
LIN {X 0,Y 18.059,Z 443.525,A -85,B 0,C 180,E1 -29686.696,E2 -29686.696} C_VEL
LIN {X 0,Y 9.062,Z 446.949,A -85,B 0,C 180,E1 -29660.906,E2 -29660.906} C_VEL
LIN {X 0,Y 6.524,Z 448.799,A -85,B 0,C 180,E1 -29610.043,E2 -29610.043} C_VEL
LIN {X 0,Y 9.043,Z 450.149,A -85,B 0,C 180,E1 -29559.049,E2 -29559.049} C_VEL
LIN {X 0,Y 14.774,Z 451.212,A -85,B 0,C 180,E1 -29538.001,E2 -29538.001} C_VEL
LIN {X 0,Y 14.268,Z 450.99,A -85,B 0,C 180,E1 -29530.006,E2 -29530.006} C_VEL
LIN {X 0,Y 5.774,Z 448.127,A -85,B 0,C 180,E1 -29467.428,E2 -29467.428} C_VEL
LIN {X 0,Y 16.145,Z 443.268,A -85,B 0,C 180,E1 -29391.894,E2 -29391.894} C_VEL
LIN {X 0,Y 28.112,Z 438.239,A -85,B 0,C 180,E1 -29381.395,E2 -29381.395} C_VEL
LIN {X 0,Y 35.157,Z 434.796,A -85,B 0,C 180,E1 -29378.176,E2 -29378.176} C_VEL
LIN {X 0,Y 40.096,Z 432.099,A -85,B 0,C 180,E1 -29375.524,E2 -29375.524} C_VEL
LIN {X 0,Y 47.787,Z 427.327,A -85,B 0,C 180,E1 -29370.215,E2 -29370.215} C_VEL
LIN {X 0,Y 55.505,Z 422.081,A -85,B 0,C 180,E1 -29366.363,E2 -29366.363} C_VEL
LIN {X 0,Y 60.272,Z 418.628,A -85,B 0,C 180,E1 -29365.543,E2 -29365.543} C_VEL
LIN {X 0,Y 64.571,Z 415.317,A -85,B 0,C 180,E1 -29365.289,E2 -29365.289} C_VEL
LIN {X 0,Y 65.396,Z 414.632,A -85,B 0,C 180,E1 -29358.801,E2 -29358.801} C_VEL
LIN {X 0,Y 65.788,Z 414.447,A -85,B 0,C 180,E1 -29355.946,E2 -29355.946} C_VEL
LIN {X 0,Y 66.134,Z 414.546,A -85,B 0,C 180,E1 -29352.264,E2 -29352.264} C_VEL
LIN {X 0,Y 64.263,Z 416.336,A -85,B 0,C 180,E1 -29350.153,E2 -29350.153} C_VEL
LIN {X 0,Y 51.717,Z 425.294,A -85,B 0,C 180,E1 -29349.83,E2 -29349.83} C_VEL
LIN {X 0,Y 37.663,Z 433.482,A -85,B 0,C 180,E1 -29349.778,E2 -29349.778} C_VEL
LIN {X 0,Y 24.957,Z 439.522,A -85,B 0,C 180,E1 -29349.659,E2 -29349.659} C_VEL
LIN {X 0,Y 10.721,Z 444.831,A -85,B 0,C 180,E1 -29350.333,E2 -29350.333} C_VEL
LIN {X 0,Y 7.172,Z 445.913,A -85,B 0,C 180,E1 -29351.32,E2 -29351.32} C_VEL
LIN {X 0,Y 7.545,Z 445.72,A -85,B 0,C 180,E1 -29361.235,E2 -29361.235} C_VEL
LIN {X 0,Y 19.82,Z 441.29,A -85,B 0,C 180,E1 -29366.586,E2 -29366.586} C_VEL
LIN {X 0,Y 31.471,Z 436.145,A -85,B 0,C 180,E1 -29366.693,E2 -29366.693} C_VEL
LIN {X 0,Y 45.022,Z 428.811,A -85,B 0,C 180,E1 -29366.143,E2 -29366.143} C_VEL
LIN {X 0,Y 58.448,Z 419.966,A -85,B 0,C 180,E1 -29365.59,E2 -29365.59} C_VEL
LIN {X 0,Y 60.272,Z 418.628,A -85,B 0,C 180,E1 -29365.543,E2 -29365.543} C_VEL
LIN {X 0,Y 60.267,Z 418.603,A -85,B 0,C 180,E1 -29364.574,E2 -29364.574} C_VEL
LIN {X 0,Y 58.9,Z 419.579,A -85,B 0,C 180,E1 -29362.765,E2 -29362.765} C_VEL
LIN {X 0,Y 54.973,Z 422.389,A -85,B 0,C 180,E1 -29359.087,E2 -29359.087} C_VEL
LIN {X 0,Y 52.509,Z 424.162,A -85,B 0,C 180,E1 -29357.412,E2 -29357.412} C_VEL
LIN {X 0,Y 51.641,Z 424.717,A -85,B 0,C 180,E1 -29357.683,E2 -29357.683} C_VEL
LIN {X 0,Y 51.732,Z 424.646,A -85,B 0,C 180,E1 -29357.998,E2 -29357.998} C_VEL
LIN {X 0,Y 59.368,Z 419.283,A -85,B 0,C 180,E1 -29358.717,E2 -29358.717} C_VEL
LIN {X 0,Y 59.897,Z 418.92,A -85,B 0,C 180,E1 -29357.564,E2 -29357.564} C_VEL
LIN {X 0,Y 58.774,Z 419.804,A -85,B 0,C 180,E1 -29356.924,E2 -29356.924} C_VEL
LIN {X 0,Y 51.641,Z 424.717,A -85,B 0,C 180,E1 -29357.683,E2 -29357.683} C_VEL
LIN {X 0,Y 50.754,Z 426.382,A -85,B 0,C 180,E1 -29357.798,E2 -29357.798} C_VEL
LIN {X 0,Y 50.754,Z 600,A -85,B 0,C 180,E1 -29357.798,E2 -29357.798} C_VEL
LIN {X 0,Y 50.754,Z 600,A -85,B 0,C 180,E1 -29357.798,E2 -29357.798}

QRS_NEXT_CUT()

QRS_NEXT()
QRS_HOME()

END
